PROGRAM MAIN
VAR
	fbSubject 			: FB_SubjectNew;
	fbObserver1 		: FB_Observer;
	fbObserver2 		: FB_Observer;
	
	bAttachObserver1	: BOOL;
	bAttachObserver2	: BOOL;

	bDetachObserver1	: BOOL;
	bDetachObserver2	: BOOL;
END_VAR

fbSubject();

IF (bAttachObserver1) THEN
	fbSubject.Attach(fbObserver1);
	bAttachObserver1 := FALSE;
END_IF

IF (bAttachObserver2) THEN
	fbSubject.Attach(fbObserver2);
	bAttachObserver2 := FALSE;
END_IF

IF (bDetachObserver1) THEN
	fbSubject.Detach(fbObserver1);
	bDetachObserver1 := FALSE;
END_IF

IF (bDetachObserver2) THEN
	fbSubject.Detach(fbObserver2);
	bDetachObserver2 := FALSE;
END_IF

END_PROGRAM

(* stored: Version 1.1.0.1, ProductVersion 3.1.4022.10
   POU MAIN: Id {d8d017fc-ecbd-440f-9cc9-45942ef857e5}, SpecialFunc None *)
